FUNCTION_BLOCK AlPgnTxNew8B_REQ (* Send data whenever a REQ (J1939 network event) occurs with Callback *)
  (* Standard: 61499-2 *)
  (* Version 1.0, 2025-09-04, franz *)
  PACKAGE isobus::pgn::tx;
  IMPORT isobus::pgn::ISONETEVENT_T;
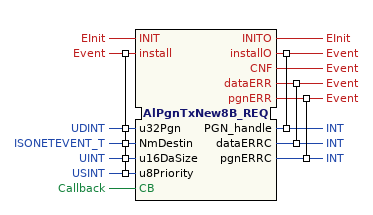
  EVENT_INPUT
    INIT : EInit; (* Service Initialization *)
    install WITH u32Pgn, NmDestin, u16DaSize, u8Priority; (* installs a Transmit PGN (TX) *)
  END_EVENT
  EVENT_OUTPUT
    INITO : EInit; (* Initialization Confirm *)
    installO WITH PGN_handle; (* install Done *)
    CNF; (* Data was sent *)
    dataERR WITH dataERRC;
    pgnERR WITH pgnERRC;
  END_EVENT
  VAR_INPUT
    u32Pgn : UDINT; (* PGN - Range: 0 - 0x3FFFF *)
    NmDestin : isobus::pgn::ISONETEVENT_T; (* Define the Communication Partner *)
    u16DaSize : UINT; (* Data length of this PGN (0..8) *)
    u8Priority : USINT := 7; (* Default priority of this PGN (0..7) 0=highest *)
  END_VAR
  VAR_OUTPUT
    PGN_handle : INT; (* PGN-handle on success, HANDLE_UNVALID in case of an error *)
    dataERRC : INT; (* dataERR error Code *)
    pgnERRC : INT; (* pgnERR error Code *)
  END_VAR
  SOCKETS
    CB : isobus::pgn::tx::Callback;
  END_SOCKETS
END_FUNCTION_BLOCK
